Staubli VAL3: VelocityCmd.pjx

--- VelocityCmd.pjx ---
Parameters version=s7.8.1 stackSize=5000 millimeterUnit=true
Program file=start.pgx
Program file=stop.pgx
Data file=VelocityCmd.dtx

--- VelocityCmd.dtx ---
public num nSeq
public num nVelVec[6]
public num nCmdType
